//returns true if part of the "ETHIP" GVL List.
FUNCTION F_Check_Symbol_In_ETHIP : BOOL
VAR_INPUT
    sSymbolName : STRING;
END_VAR
VAR
END_VAR

IF LEFT(sSymbolName, 6) = 'ETHIP.' THEN
    F_Check_Symbol_In_ETHIP := TRUE;
ELSE
    F_Check_Symbol_In_ETHIP := FALSE;
END_IF

END_FUNCTION

(* stored: Version 1.1.0.1, ProductVersion 3.1.4024.12
   POU F_Check_Symbol_In_ETHIP: Id {b164eced-4e27-4d9a-8f28-d3d306970ac3}, SpecialFunc None *)
